PROGRAM MAIN
VAR
	i: INT;
	error_counter: INT := 0;
	time_out_counter: UDINT :=0;
	num_of_axis: INT := 7;
	axis_index: INT := 0;
	online_counter: UDINT := 0;
	write_counter: UDINT := 1;
	
	fVel_Arm : ARRAY[1..7] OF LREAL := [7(0)];
	fAcc_Arm : ARRAY[1..7] OF LREAL := [7(0)];
	fDec_Arm : ARRAY[1..7] OF LREAL := [7(0)];
	fJerk_Arm : ARRAY[1..7] OF LREAL := [7(0)];
	fPos_Yaw : LREAL ;
	fDir_Arm : ARRAY[1..7] OF MC_DIRECTION;
	
	MC_Move_1_Absolute: ARRAY[1..7] OF MC_MoveAbsolute;
	MC_Move_2_Absolute: ARRAY[1..7] OF MC_MoveAbsolute;
	bMove_1_Arm_Abs: BOOL := FALSE;
	bMove_2_Arm_Abs: BOOL := FALSE;
	
	nState: INT := 930;
	bSetPos_Yaw: BOOL;
	MC_SetPosition_Yaw: MC_SetPosition;
END_VAR

ACT_Power();
//Mov_Absolute();

//IF state_INIT THEN
//	ACT_LimitSwitch();
//ELSE
	
IF fLastTimeStamp <> 0 AND (fActTimeStamp - fLastTimeStamp) = 0 THEN
	time_out_counter := time_out_counter + 1;
ELSE
	time_out_counter := 0;
END_IF

IF time_out_counter > max_time_out THEN
	state_TIMEOUT := TRUE;
	state_HALT := TRUE;
	fLastTimeStamp:= 0;
	fActTimeStamp:= 0;
	time_out_counter := 0;
	FOR axis_index:=1 TO num_of_axis DO
		f_Halt_Dec_Arm[axis_index] := EksenArm[axis_index].NcToPlc.ActAcc * 5;
		fVel_Arm[axis_index] := 0.0;
		fAcc_Arm[axis_index] := 0.0;
		fDec_Arm[axis_index] := 0.0;
	END_FOR
ELSE
	//////////////// SET DIRECTION \\\\\\\\\\\\\\\\\\\\\\

	FOR axis_index:=1 TO num_of_axis DO
		IF fGoalVel_Arm[axis_index] < 0 THEN
			fDir_Arm[axis_index] := MC_Negative_Direction;
		ELSE
			fDir_Arm[axis_index] := MC_Positive_Direction;
		END_IF
	END_FOR
	
	//////////////// SET PARAMETERS \\\\\\\\\\\\\\\\\\\\\\
	
	FOR axis_index:=1 TO num_of_axis DO	
		fVel_Arm[axis_index] := ABS(fGoalVel_Arm[axis_index]);
		fAcc_Arm[axis_index] := ABS(fGoalAcc_Arm[axis_index]);
		fDec_Arm[axis_index] := ABS(fGoalAcc_Arm[axis_index]);
	END_FOR	
END_IF

//////////////// FILL UP JOINT STATES \\\\\\\\\\\\\\\\\\\\\\

FOR axis_index:=1 TO num_of_axis DO	
	fActPose_Arm[axis_index] := EksenArm[axis_index].NcToPlc.ActPos;
	fActVel_Arm[axis_index] := EksenArm[axis_index].NcToPlc.ActVelo;
END_FOR	

//////////////// SAVE DATA \\\\\\\\\\\\\\\\\\\\\\

IF SAVE_DATA THEN
	IF (online_counter MOD 25) = 0 THEN
		FOR i:=1 TO 7 DO
			csvActPos[write_counter, i] := EksenArm[i].NcToPlc.ActPos;
			csvActVel[write_counter, i] := EksenArm[i].NcToPlc.ActVelo;
			csvGoalPos[write_counter, i] := fGoalPos_Arm[i];
			csvGoalVel[write_counter, i] := fGoalVel_Arm[i];
		END_FOR
		write_counter:= write_counter + 1;
	END_IF
	online_counter:= online_counter + 1;	
END_IF

////////////// CHECK ERROR STATE \\\\\\\\\\\\\\\\\\\\\\

//FOR error_counter:=1 TO num_of_axis DO
//	IF PowerAxisArm[error_counter].ErrorID <> 0 THEN
//		Error_latch[error_counter] := 100;
//		bMove_1_Arm := FALSE;
//		bMove_2_Arm := FALSE;
//		bRunBlocks := FALSE;
//		state_HALT := TRUE;
//		FOR halt_counter:=1 TO num_of_axis DO
//			f_Halt_Dec_Arm[halt_counter] := EksenArm[halt_counter].NcToPlc.ActAcc * 5;
//		END_FOR
//	END_IF
//END_FOR


////////////// SWITCH MOTION BLOCKS \\\\\\\\\\\\\\\\\\\\\\

IF bMove_1_Arm THEN
	bMove_1_Arm := FALSE;
	bMove_2_Arm := TRUE;
ELSE
	bMove_1_Arm := TRUE;
	bMove_2_Arm := FALSE;
END_IF


fLastTimeStamp := fActTimeStamp;

//END_IF

ACTION ACT_LimitSwitch:
IF EksenArm[2].NcToPlc.ActPos < 20.0 THEN
	Main.fVel_Arm[2] := 5.0;
	Main.fDir_Arm[2] := MC_Positive_Direction;
ELSE
	fVel_Arm[2] := 0.0;

	IF NOT bLimitSwitch THEN	
		fVel_Arm[7] := 20.0;
		Main.fDir_Arm[7] := MC_Negative_Direction;
	ELSE
		Main.bSetPos_Yaw := TRUE;	
		fVel_Arm[7] := 0.0;
		Mc_SetPosition_Yaw.Position := -120.0;
		state_INIT := FALSE;
	END_IF
END_IF

IF bMove_1_Arm THEN
	bMove_1_Arm := FALSE;
	bMove_2_Arm := TRUE;
ELSE
	bMove_1_Arm := TRUE;
	bMove_2_Arm := FALSE;
END_IF
END_ACTION

ACTION ACT_Power:
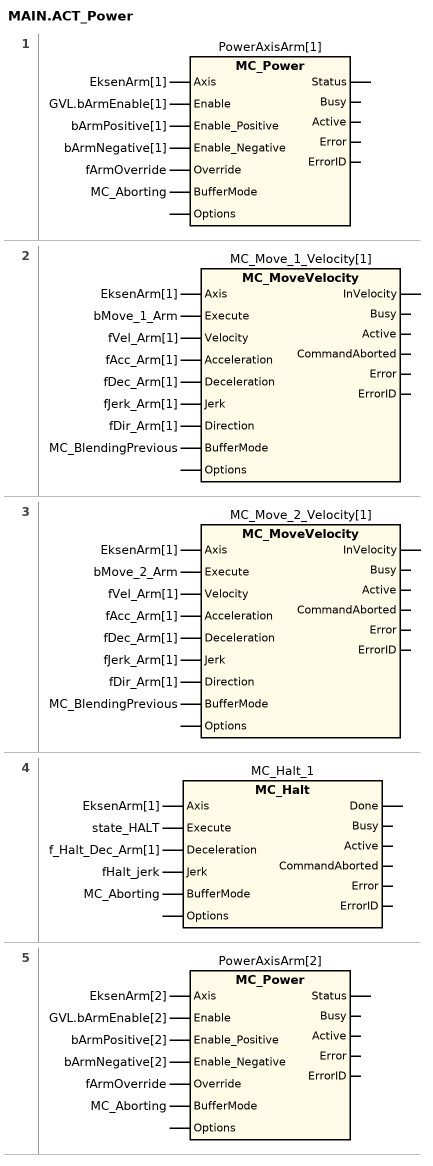
// NETWORK 1
PowerAxisArm[1](
    Axis := EksenArm[1],
    Enable := GVL.bArmEnable[1],
    Enable_Positive := bArmPositive[1],
    Enable_Negative := bArmNegative[1],
    Override := fArmOverride,
    BufferMode := MC_Aborting); // MC_Power

// NETWORK 2
MC_Move_1_Velocity[1](
    Axis := EksenArm[1],
    Execute := bMove_1_Arm,
    Velocity := fVel_Arm[1],
    Acceleration := fAcc_Arm[1],
    Deceleration := fDec_Arm[1],
    Jerk := fJerk_Arm[1],
    Direction := fDir_Arm[1],
    BufferMode := MC_BlendingPrevious); // MC_MoveVelocity

// NETWORK 3
MC_Move_2_Velocity[1](
    Axis := EksenArm[1],
    Execute := bMove_2_Arm,
    Velocity := fVel_Arm[1],
    Acceleration := fAcc_Arm[1],
    Deceleration := fDec_Arm[1],
    Jerk := fJerk_Arm[1],
    Direction := fDir_Arm[1],
    BufferMode := MC_BlendingPrevious); // MC_MoveVelocity

// NETWORK 4
MC_Halt_1(
    Axis := EksenArm[1],
    Execute := state_HALT,
    Deceleration := f_Halt_Dec_Arm[1],
    Jerk := fHalt_jerk,
    BufferMode := MC_Aborting); // MC_Halt

// NETWORK 5
PowerAxisArm[2](
    Axis := EksenArm[2],
    Enable := GVL.bArmEnable[2],
    Enable_Positive := bArmPositive[2],
    Enable_Negative := bArmNegative[2],
    Override := fArmOverride,
    BufferMode := MC_Aborting); // MC_Power

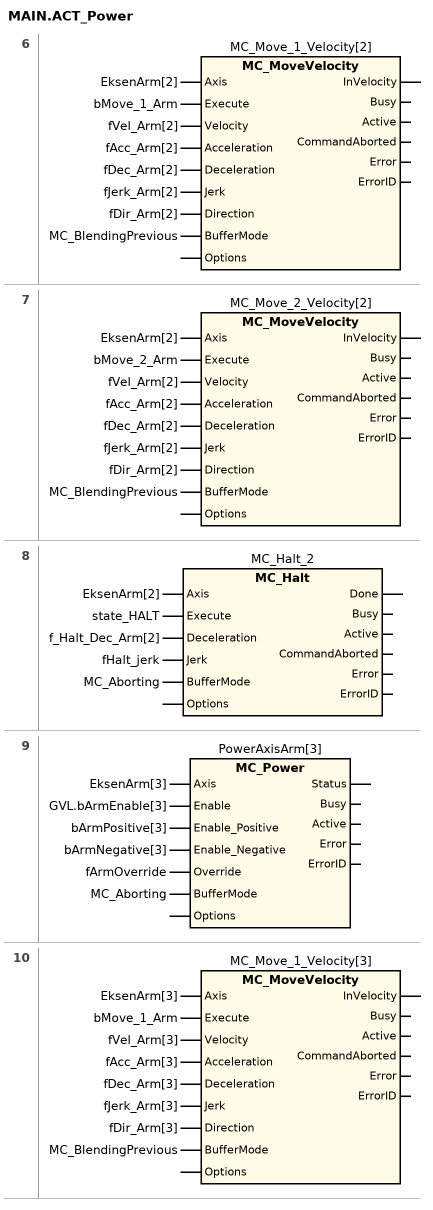
// NETWORK 6
MC_Move_1_Velocity[2](
    Axis := EksenArm[2],
    Execute := bMove_1_Arm,
    Velocity := fVel_Arm[2],
    Acceleration := fAcc_Arm[2],
    Deceleration := fDec_Arm[2],
    Jerk := fJerk_Arm[2],
    Direction := fDir_Arm[2],
    BufferMode := MC_BlendingPrevious); // MC_MoveVelocity

// NETWORK 7
MC_Move_2_Velocity[2](
    Axis := EksenArm[2],
    Execute := bMove_2_Arm,
    Velocity := fVel_Arm[2],
    Acceleration := fAcc_Arm[2],
    Deceleration := fDec_Arm[2],
    Jerk := fJerk_Arm[2],
    Direction := fDir_Arm[2],
    BufferMode := MC_BlendingPrevious); // MC_MoveVelocity

// NETWORK 8
MC_Halt_2(
    Axis := EksenArm[2],
    Execute := state_HALT,
    Deceleration := f_Halt_Dec_Arm[2],
    Jerk := fHalt_jerk,
    BufferMode := MC_Aborting); // MC_Halt

// NETWORK 9
PowerAxisArm[3](
    Axis := EksenArm[3],
    Enable := GVL.bArmEnable[3],
    Enable_Positive := bArmPositive[3],
    Enable_Negative := bArmNegative[3],
    Override := fArmOverride,
    BufferMode := MC_Aborting); // MC_Power

// NETWORK 10
MC_Move_1_Velocity[3](
    Axis := EksenArm[3],
    Execute := bMove_1_Arm,
    Velocity := fVel_Arm[3],
    Acceleration := fAcc_Arm[3],
    Deceleration := fDec_Arm[3],
    Jerk := fJerk_Arm[3],
    Direction := fDir_Arm[3],
    BufferMode := MC_BlendingPrevious); // MC_MoveVelocity

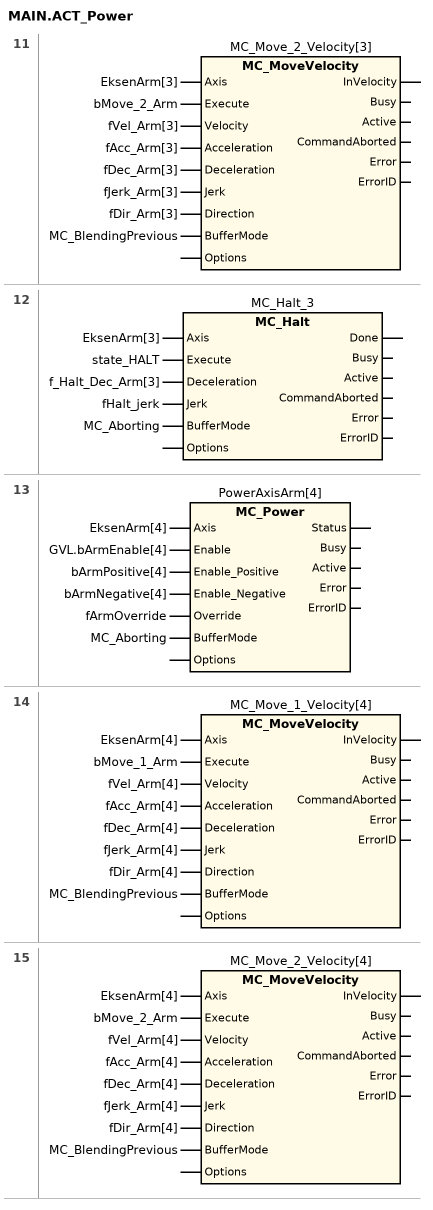
// NETWORK 11
MC_Move_2_Velocity[3](
    Axis := EksenArm[3],
    Execute := bMove_2_Arm,
    Velocity := fVel_Arm[3],
    Acceleration := fAcc_Arm[3],
    Deceleration := fDec_Arm[3],
    Jerk := fJerk_Arm[3],
    Direction := fDir_Arm[3],
    BufferMode := MC_BlendingPrevious); // MC_MoveVelocity

// NETWORK 12
MC_Halt_3(
    Axis := EksenArm[3],
    Execute := state_HALT,
    Deceleration := f_Halt_Dec_Arm[3],
    Jerk := fHalt_jerk,
    BufferMode := MC_Aborting); // MC_Halt

// NETWORK 13
PowerAxisArm[4](
    Axis := EksenArm[4],
    Enable := GVL.bArmEnable[4],
    Enable_Positive := bArmPositive[4],
    Enable_Negative := bArmNegative[4],
    Override := fArmOverride,
    BufferMode := MC_Aborting); // MC_Power

// NETWORK 14
MC_Move_1_Velocity[4](
    Axis := EksenArm[4],
    Execute := bMove_1_Arm,
    Velocity := fVel_Arm[4],
    Acceleration := fAcc_Arm[4],
    Deceleration := fDec_Arm[4],
    Jerk := fJerk_Arm[4],
    Direction := fDir_Arm[4],
    BufferMode := MC_BlendingPrevious); // MC_MoveVelocity

// NETWORK 15
MC_Move_2_Velocity[4](
    Axis := EksenArm[4],
    Execute := bMove_2_Arm,
    Velocity := fVel_Arm[4],
    Acceleration := fAcc_Arm[4],
    Deceleration := fDec_Arm[4],
    Jerk := fJerk_Arm[4],
    Direction := fDir_Arm[4],
    BufferMode := MC_BlendingPrevious); // MC_MoveVelocity

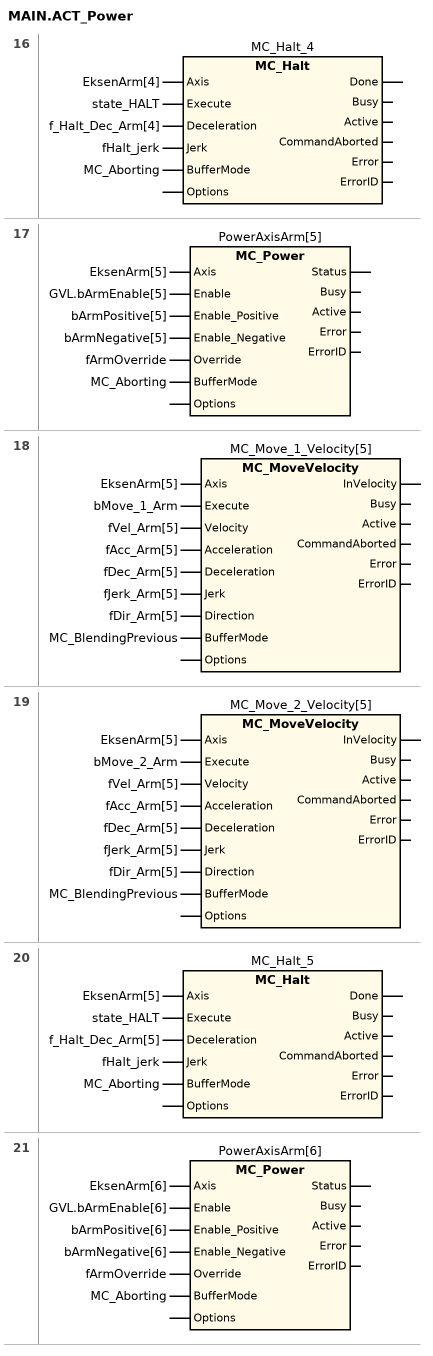
// NETWORK 16
MC_Halt_4(
    Axis := EksenArm[4],
    Execute := state_HALT,
    Deceleration := f_Halt_Dec_Arm[4],
    Jerk := fHalt_jerk,
    BufferMode := MC_Aborting); // MC_Halt

// NETWORK 17
PowerAxisArm[5](
    Axis := EksenArm[5],
    Enable := GVL.bArmEnable[5],
    Enable_Positive := bArmPositive[5],
    Enable_Negative := bArmNegative[5],
    Override := fArmOverride,
    BufferMode := MC_Aborting); // MC_Power

// NETWORK 18
MC_Move_1_Velocity[5](
    Axis := EksenArm[5],
    Execute := bMove_1_Arm,
    Velocity := fVel_Arm[5],
    Acceleration := fAcc_Arm[5],
    Deceleration := fDec_Arm[5],
    Jerk := fJerk_Arm[5],
    Direction := fDir_Arm[5],
    BufferMode := MC_BlendingPrevious); // MC_MoveVelocity

// NETWORK 19
MC_Move_2_Velocity[5](
    Axis := EksenArm[5],
    Execute := bMove_2_Arm,
    Velocity := fVel_Arm[5],
    Acceleration := fAcc_Arm[5],
    Deceleration := fDec_Arm[5],
    Jerk := fJerk_Arm[5],
    Direction := fDir_Arm[5],
    BufferMode := MC_BlendingPrevious); // MC_MoveVelocity

// NETWORK 20
MC_Halt_5(
    Axis := EksenArm[5],
    Execute := state_HALT,
    Deceleration := f_Halt_Dec_Arm[5],
    Jerk := fHalt_jerk,
    BufferMode := MC_Aborting); // MC_Halt

// NETWORK 21
PowerAxisArm[6](
    Axis := EksenArm[6],
    Enable := GVL.bArmEnable[6],
    Enable_Positive := bArmPositive[6],
    Enable_Negative := bArmNegative[6],
    Override := fArmOverride,
    BufferMode := MC_Aborting); // MC_Power

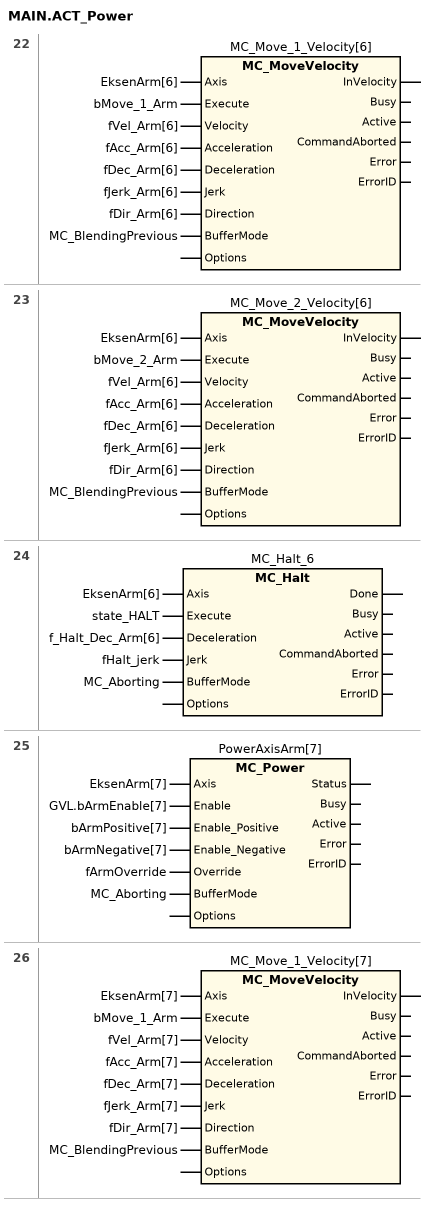
// NETWORK 22
MC_Move_1_Velocity[6](
    Axis := EksenArm[6],
    Execute := bMove_1_Arm,
    Velocity := fVel_Arm[6],
    Acceleration := fAcc_Arm[6],
    Deceleration := fDec_Arm[6],
    Jerk := fJerk_Arm[6],
    Direction := fDir_Arm[6],
    BufferMode := MC_BlendingPrevious); // MC_MoveVelocity

// NETWORK 23
MC_Move_2_Velocity[6](
    Axis := EksenArm[6],
    Execute := bMove_2_Arm,
    Velocity := fVel_Arm[6],
    Acceleration := fAcc_Arm[6],
    Deceleration := fDec_Arm[6],
    Jerk := fJerk_Arm[6],
    Direction := fDir_Arm[6],
    BufferMode := MC_BlendingPrevious); // MC_MoveVelocity

// NETWORK 24
MC_Halt_6(
    Axis := EksenArm[6],
    Execute := state_HALT,
    Deceleration := f_Halt_Dec_Arm[6],
    Jerk := fHalt_jerk,
    BufferMode := MC_Aborting); // MC_Halt

// NETWORK 25
PowerAxisArm[7](
    Axis := EksenArm[7],
    Enable := GVL.bArmEnable[7],
    Enable_Positive := bArmPositive[7],
    Enable_Negative := bArmNegative[7],
    Override := fArmOverride,
    BufferMode := MC_Aborting); // MC_Power

// NETWORK 26
MC_Move_1_Velocity[7](
    Axis := EksenArm[7],
    Execute := bMove_1_Arm,
    Velocity := fVel_Arm[7],
    Acceleration := fAcc_Arm[7],
    Deceleration := fDec_Arm[7],
    Jerk := fJerk_Arm[7],
    Direction := fDir_Arm[7],
    BufferMode := MC_BlendingPrevious); // MC_MoveVelocity

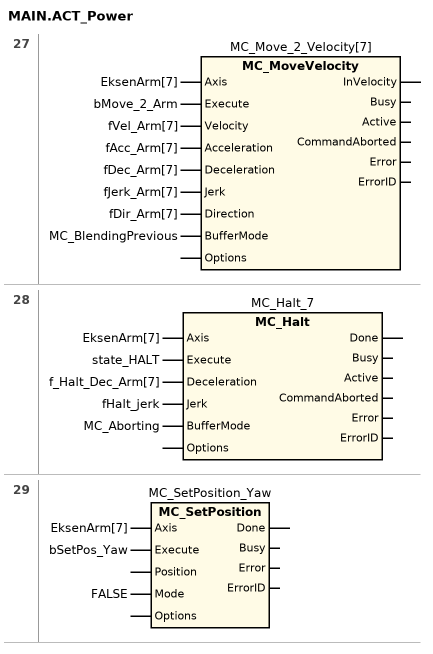
// NETWORK 27
MC_Move_2_Velocity[7](
    Axis := EksenArm[7],
    Execute := bMove_2_Arm,
    Velocity := fVel_Arm[7],
    Acceleration := fAcc_Arm[7],
    Deceleration := fDec_Arm[7],
    Jerk := fJerk_Arm[7],
    Direction := fDir_Arm[7],
    BufferMode := MC_BlendingPrevious); // MC_MoveVelocity

// NETWORK 28
MC_Halt_7(
    Axis := EksenArm[7],
    Execute := state_HALT,
    Deceleration := f_Halt_Dec_Arm[7],
    Jerk := fHalt_jerk,
    BufferMode := MC_Aborting); // MC_Halt

// NETWORK 29
MC_SetPosition_Yaw(Axis := EksenArm[7], Execute := bSetPos_Yaw, Mode := FALSE); // MC_SetPosition
END_ACTION

ACTION Mov_Absolute:
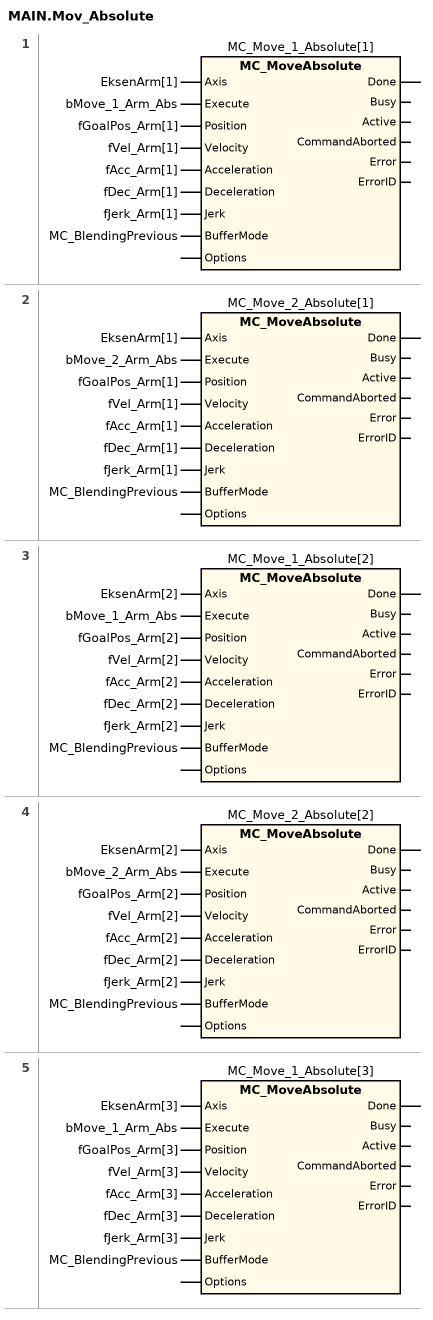
// NETWORK 1
MC_Move_1_Absolute[1](
    Axis := EksenArm[1],
    Execute := bMove_1_Arm_Abs,
    Position := fGoalPos_Arm[1],
    Velocity := fVel_Arm[1],
    Acceleration := fAcc_Arm[1],
    Deceleration := fDec_Arm[1],
    Jerk := fJerk_Arm[1],
    BufferMode := MC_BlendingPrevious); // MC_MoveAbsolute

// NETWORK 2
MC_Move_2_Absolute[1](
    Axis := EksenArm[1],
    Execute := bMove_2_Arm_Abs,
    Position := fGoalPos_Arm[1],
    Velocity := fVel_Arm[1],
    Acceleration := fAcc_Arm[1],
    Deceleration := fDec_Arm[1],
    Jerk := fJerk_Arm[1],
    BufferMode := MC_BlendingPrevious); // MC_MoveAbsolute

// NETWORK 3
MC_Move_1_Absolute[2](
    Axis := EksenArm[2],
    Execute := bMove_1_Arm_Abs,
    Position := fGoalPos_Arm[2],
    Velocity := fVel_Arm[2],
    Acceleration := fAcc_Arm[2],
    Deceleration := fDec_Arm[2],
    Jerk := fJerk_Arm[2],
    BufferMode := MC_BlendingPrevious); // MC_MoveAbsolute

// NETWORK 4
MC_Move_2_Absolute[2](
    Axis := EksenArm[2],
    Execute := bMove_2_Arm_Abs,
    Position := fGoalPos_Arm[2],
    Velocity := fVel_Arm[2],
    Acceleration := fAcc_Arm[2],
    Deceleration := fDec_Arm[2],
    Jerk := fJerk_Arm[2],
    BufferMode := MC_BlendingPrevious); // MC_MoveAbsolute

// NETWORK 5
MC_Move_1_Absolute[3](
    Axis := EksenArm[3],
    Execute := bMove_1_Arm_Abs,
    Position := fGoalPos_Arm[3],
    Velocity := fVel_Arm[3],
    Acceleration := fAcc_Arm[3],
    Deceleration := fDec_Arm[3],
    Jerk := fJerk_Arm[3],
    BufferMode := MC_BlendingPrevious); // MC_MoveAbsolute

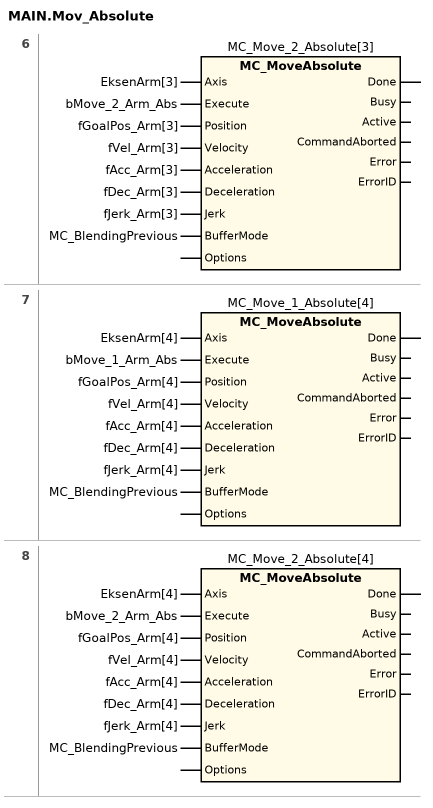
// NETWORK 6
MC_Move_2_Absolute[3](
    Axis := EksenArm[3],
    Execute := bMove_2_Arm_Abs,
    Position := fGoalPos_Arm[3],
    Velocity := fVel_Arm[3],
    Acceleration := fAcc_Arm[3],
    Deceleration := fDec_Arm[3],
    Jerk := fJerk_Arm[3],
    BufferMode := MC_BlendingPrevious); // MC_MoveAbsolute

// NETWORK 7
MC_Move_1_Absolute[4](
    Axis := EksenArm[4],
    Execute := bMove_1_Arm_Abs,
    Position := fGoalPos_Arm[4],
    Velocity := fVel_Arm[4],
    Acceleration := fAcc_Arm[4],
    Deceleration := fDec_Arm[4],
    Jerk := fJerk_Arm[4],
    BufferMode := MC_BlendingPrevious); // MC_MoveAbsolute

// NETWORK 8
MC_Move_2_Absolute[4](
    Axis := EksenArm[4],
    Execute := bMove_2_Arm_Abs,
    Position := fGoalPos_Arm[4],
    Velocity := fVel_Arm[4],
    Acceleration := fAcc_Arm[4],
    Deceleration := fDec_Arm[4],
    Jerk := fJerk_Arm[4],
    BufferMode := MC_BlendingPrevious); // MC_MoveAbsolute
END_ACTION

END_PROGRAM

(* stored: Version 1.1.0.1, ProductVersion 3.1.4024.9
   POU MAIN: Id {2cdeb687-4fce-4d88-bc1f-27e6f03e98e2}, SpecialFunc None
   Action ACT_LimitSwitch: Id {e0562fdb-77f8-45bc-bb7a-6ff33d4cb15b}
   Action ACT_Power: Id {4c9ef814-d7e6-4c47-b37a-7bb54b9a6811}
   Action Mov_Absolute: Id {9d353036-170d-406a-8ed6-8341038067ba} *)
